// TwinCAT 3 PLC project StrawberryPLC
// ProgramVersion: 3.1.4023.0
// libraries:
//   Tc2_Standard, * (Beckhoff Automation GmbH)
//   Tc2_System, * (Beckhoff Automation GmbH)
//   Tc3_Module, * (Beckhoff Automation GmbH)
//   Tc3_Vision, * (Beckhoff Automation GmbH)
// project tree:
//   / PlcTask.TcTTO
//   POUs/ FB_ConvertColourSpace.TcPOU, FindRed.TcPOU, F_ConvertColorSpaceST.TcPOU, F_DrawOrientation.TcPOU, F_GetOrientationST.TcPOU, MAIN.TcPOU
// real-time tasks:
//   TASK PlcTask: cycle T#10ms, priority 20, ADS port 350
//   TASK VnTask ImgAcq (FileSource1): cycle T#10ms, priority 5, ADS port 351

CONFIGURATION StrawberryPLC
    RESOURCE PLC ON TwinCAT3
        TASK PlcTask(INTERVAL := T#10ms, PRIORITY := 20);
        PROGRAM MAIN WITH PlcTask : MAIN;
    END_RESOURCE
END_CONFIGURATION

// ---- POUs/MAIN.TcPOU
PROGRAM MAIN
VAR
	hr				: HRESULT; //each camera will need a individual HRESULT variable
	fbCamera		: FB_VN_FileSourceControl;
//this variable links the plc to our vision node// can be either FB_VN_GevCameraControl or "  "_FileSourceControl
	eState			: ETcVnCameraState; //Takes current state of the camera
	
	ipImageIn		: ITcVnImage; //Raw Image data and meta data. can't be seen by humans
	ipImageInDisp	: ITcVnDisplayableImage; //Converts raw data and meta data to something displayable which can be used in an HMI
	ipImageWork		: ITcVnImage;
	ipImageResult	: ITcVnImage;
	ipImageResultDisp	: ITcVnDisplayableImage;
	
	ipImageColorMap_Red: ITcVnImage;
	ipImageColorMap_Red2: ITcVnImage;
	
	ipImageColorMapDisp_Red2: ITcVnDisplayableImage;
	
	ipImageColorMap_Red3: ITcVnImage;
	ipImageColorMapDisp_Red3: ITcVnDisplayableImage;
	// lower mask
	aColorLow_Red	: TcVnVector4_LREAL := [0,50,50];
	aColorUpper_Red	: TcVnVector4_LREAL := [10,255,255];
	// upper mask
	aColorLow_Red2	: TcVnVector4_LREAL := [170,50,50];
	aColorUpper_Red2: TcVnVector4_LREAL := [180,255,255];
	
	ipImageOnlyStawberry: ITcVnImage;
	
	ipContourList	: ITcVnContainer;
	ipIterator		: ITcVnForwardIterator;
	ipContour		: ITcVnContainer;
	
	aColor_RED		: TcVnVector4_LREAL:= [255,0,0];
	
	// My own code
	ColourConverter : FB_ConvertColourSpace;
	
	
	fElement     : REAL;
END_VAR

CASE eState OF
	//-------------------------------------------------------------------------------------------------------
	TCVN_CS_INITIAL, TCVN_CS_OPENING, TCVN_CS_OPENED, TCVN_CS_STARTACQUISITION:
		hr := fbCamera.StartAcquisition();
	//-------------------------------------------------------------------------------------------------------
	TCVN_CS_ERROR:
		hr := fbCamera.Reset();
	//---------------------------------------------------------------------------------------------------------
	TCVN_CS_ACQUIRING:
		hr := fbCamera.GetCurrentImage(ipImageIN);
		IF SUCCEEDED(hr) AND ipImageIn <> 0 THEN
			//
		hr := F_VN_CopyImage(ipImageIn, ipImageResult,hr);
		hr := F_VN_CopyIntoDisplayableImage(ipImageIn, ipImageInDisp, hr);
		// blur image
		hr := F_VN_GaussianFilter(ipImageIn,ipImageWork,51,51,hr);
		//------------------------------------------------------------------------------------------------------
		// convert RGB space to HSV
		hr := F_VN_ConvertColorSpace(ipImageWork, ipImageWork, TCVN_CST_RGB_TO_HSV, hr);
		//ColourConverter(hr_internal:=hr, ipImageIn := ipImageIn, ColourSpaceType:='GRAY', ipImageOut=>ipImageWork);
		//ColourConverter(); this is only need if i don't do the code above
		
		//hr := F_VN_CopyIntoDisplayableImage(ipImageWork,ipImageColorMapDisp_Red2,hr);
		//------------------------------------------------------------------------------------------------------
		//Creating first mask
		hr := F_VN_CheckColorRange(ipImageWork, ipImageColorMap_Red,aColorLow_Red,aColorUpper_Red,hr);
		//creating second mask
		hr := F_VN_CheckColorRange(ipImageWork, ipImageColorMap_Red2,aColorLow_Red2,aColorUpper_Red2,hr);
		//Adding masks together
		hr := F_VN_BitwiseOrImages(ipImageColorMap_Red,ipImageColorMap_Red2,ipImageColorMap_Red3,hr);
		//I think the reason why F_VN_BitwiseAndImages didn't work on the coloured image 
		//is because the colour is an array while the mask is a single bit
		//-----------------------------------------------------------------------------------------------
		hr := F_VN_ConvertColorSpace(ipImageIn, ipImageWork, TCVN_CST_RGB_TO_GRAY, hr);
		hr := F_VN_GaussianFilter(ipImageWork,ipImageWork,51,51,hr);
		hr := F_VN_CopyIntoDisplayableImage(ipImageWork,ipImageColorMapDisp_Red2,hr);
		hr := F_VN_BitwiseAndImages(ipImageColorMap_Red3,ipImageWork,ipImageOnlyStawberry,hr);
		
		hr := F_VN_CannyEdgeDetection(ipImageOnlyStawberry,ipImageOnlyStawberry,10,200,hr);
		
		hr := F_VN_CopyIntoDisplayableImage(ipImageOnlyStawberry,ipImageColorMapDisp_Red3,hr);
		hr := F_VN_FindContours(ipImageOnlyStawberry,ipContourList,hr);
		hr := F_VN_GetAt_REAL(ipContourList, fElement, 0, hr);
		
		
		hr := F_VN_GetForwardIterator(ipContourList, ipIterator, hr);
		
		WHILE SUCCEEDED(hr) AND_THEN ipIterator.CheckIfEnd() <> S_OK DO
			hr := F_VN_GetContainer(ipIterator, ipContour,hr);
			hr := F_VN_IncrementIterator(ipIterator,hr);
			//ADSLOGSTR(msgCtrlMask := ADSLOG_MSGTYPE_ERROR OR ADSLOG_MSGTYPE_LOG,
			//msgFmtStr := 'Container %s',
			//strArg := ipContour);
			hr := F_VN_DrawContours(ipContour, -1, ipImageResult, aColor_RED, 3,hr);
		END_WHILE
		
		hr := F_VN_CopyIntoDisplayableImage(ipImageResult,ipImageResultDisp,hr);
		END_IF
END_CASE

END_PROGRAM

// ---- POUs/FB_ConvertColourSpace.TcPOU
FUNCTION_BLOCK FB_ConvertColourSpace
VAR_INPUT
	hr_internal			: HRESULT; 
	ipImageIn		: ITcVnImage; //Only takes RGB
	ColourSpaceType	:STRING; // Only HSV or GRAY for now
END_VAR
VAR_OUTPUT
	ipImageOut		: ITcVnImage;
END_VAR
VAR
	GRAY	:STRING := 'GRAY';
	HSV		:STRING := 'HSV';
END_VAR

IF ColourSpaceType = 'GRAY' THEN
	hr_internal	:= F_VN_ConvertColorSpace(ipImageIn, ipImageOut, TCVN_CST_RGB_TO_GRAY, hr_internal	);
ELSIF ColourSpaceType = 'HSV' THEN
	hr_internal	 := F_VN_ConvertColorSpace(ipImageIn, ipImageOut, TCVN_CST_RGB_TO_HSV, hr_internal	);
END_IF

END_FUNCTION_BLOCK

// ---- POUs/FindRed.TcPOU
FUNCTION_BLOCK FindRed
VAR_INPUT 
	hr 				: HRESULT;
	ipImageIn		: ITcVnImage;
	aLowerRedBottom	: TcVnVector4_LREAL;
	aLowerRedTop		: TcVnVector4_LREAL;
	aUpperRedBottom	: TcVnVector4_LREAL;
	aUpperRedTop		: TcVnVector4_LREAL;
END_VAR
VAR_OUTPUT
	ipImageOut		: ITcVnImage; //Returns a Grey image of where the red is
END_VAR
VAR
	ipImageColorMap_Red: ITcVnImage;
	ipImageColorMap_Red2: ITcVnImage;
	ipImageColorMap_Red3: ITcVnImage;
END_VAR
VAR_IN_OUT
	
END_VAR

//Creating first mask
hr := F_VN_CheckColorRange(ipImageIn, ipImageColorMap_Red,aLowerRedBottom,aLowerRedTop,hr);
//creating second mask
hr := F_VN_CheckColorRange(ipImageIn, ipImageColorMap_Red2,aUpperRedBottom,aUpperRedTop,hr);
//Adding masks together
hr := F_VN_BitwiseOrImages(ipImageColorMap_Red,ipImageColorMap_Red2,ipImageColorMap_Red3,hr);

END_FUNCTION_BLOCK

// ---- POUs/F_ConvertColorSpaceST.TcPOU
FUNCTION F_ConvertColorSpaceST
VAR_INPUT
END_VAR
VAR
END_VAR

END_FUNCTION

// ---- POUs/F_DrawOrientation.TcPOU
FUNCTION F_DrawOrientation : HRESULT
VAR_INPUT
    ipSrcImage  : ITcVnImage;
    ipDestImage : Reference To  ITcVnImage;
    eTransform  : ETcVnColorSpaceTransform;
    hrPrev      : HRESULT;
END_VAR
VAR
	ipContourList	: ITcVnContainer;
	ipIterator		: ITcVnForwardIterator;
	ipContour		: ITcVnContainer;
	
	fArea                 :    LREAL;
	fAreaMin              :    LREAL := 100;
	fAreaMax              :    LREAL := 100000;
END_VAR

hrPrev := F_VN_FindContours(ipSrcImage,ipContourList,hrPrev);
hrPrev := F_VN_GetForwardIterator(ipContourList, ipIterator, hrPrev);

WHILE SUCCEEDED(hrPrev) AND_THEN ipIterator.CheckIfEnd() <> S_OK DO
	hrPrev := F_VN_GetContainer(ipIterator, ipContour,hrPrev);
	hrPrev := F_VN_IncrementIterator(ipIterator,hrPrev);
	
	// Filter by Area
    hrPrev := F_VN_ContourArea(ipContour, fArea, hrPrev);
	
	IF fArea > fAreaMin AND fArea < fAreaMax THEN
		hrPrev := F_GetOrientationST(
	END_IF
END_WHILE

END_FUNCTION

// ---- POUs/F_GetOrientationST.TcPOU
FUNCTION F_GetOrientationST : BOOL
VAR_INPUT
	SrcContour		: ITcVnContainer;
    ipDestImage : Reference To  ITcVnImage;
    eTransform  : ETcVnColorSpaceTransform;
    hrPrev      : HRESULT;
END_VAR
VAR
	size : ULINT;
END_VAR

size := SrcContour.GetElementNum;
//getElementNum is # of elements
//getElementSize is byte size
for

END_FUNCTION
